FUNCTION_BLOCK ReqPanelLift (* Composite Function Block Type *)
  (* Standard: 61499-2 *)
  (* Version 0.0, 6/3/2016, Andrei, nxtControl GmbH, template *)
  PACKAGE Main;
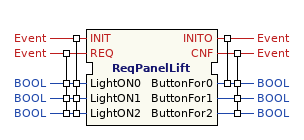
  EVENT_INPUT
    INIT WITH LightON0, LightON1, LightON2; (* Initialization Request *)
    REQ WITH LightON0, LightON1, LightON2; (* Normal Execution Request *)
  END_EVENT
  EVENT_OUTPUT
    INITO WITH ButtonFor0; (* Initialization Confirm *)
    CNF WITH ButtonFor0, ButtonFor1, ButtonFor2; (* Execution Confirmation *)
  END_EVENT
  VAR_INPUT
    LightON0 : BOOL;
    LightON1 : BOOL;
    LightON2 : BOOL;
  END_VAR
  VAR_OUTPUT
    ButtonFor0 : BOOL; (* Output event qualifier *)
    ButtonFor1 : BOOL;
    ButtonFor2 : BOOL;
  END_VAR
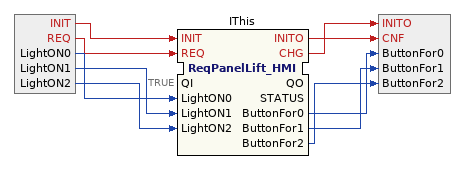
  FBS
    IThis : ReqPanelLift_HMI(QI := TRUE);
  END_FBS
  EVENT_CONNECTIONS
    INIT TO IThis.INIT;
    REQ TO IThis.REQ;
    IThis.INITO TO INITO;
    IThis.CHG TO CNF;
  END_CONNECTIONS
  DATA_CONNECTIONS
    IThis.ButtonFor0 TO ButtonFor0;
    IThis.ButtonFor1 TO ButtonFor1;
    IThis.ButtonFor2 TO ButtonFor2;
    LightON2 TO IThis.LightON2;
    LightON1 TO IThis.LightON1;
    LightON0 TO IThis.LightON0;
  END_CONNECTIONS
END_FUNCTION_BLOCK
